{attribute 'qualified_only'}
{attribute 'strict'}
{attribute 'to_string'}
TYPE nLaser_ErrorCodes :
(
	// Błędy ogólne
	NoError := 0,
	UnKnownAlarm := 53,						// Niezidentyfikowany alarm maszyny
	UnKnownLock := 54,						// Niezidentyfikowana blokada maszyny
	ProgramConfigError := 90,				// Błąd w konfiguracji programu
	LaserTCPCommunicationError := 1321		// Błąd komunikacji przez TCP z laserem
);
END_TYPE

(* stored: Version 1.1.0.1, ProductVersion 3.1.4024.15
   EnumerationTextList nLaser_ErrorCodes: Id {dc1216e8-859b-4444-9efd-96e06627c588} *)
